(* PLC project CodesysTest.project, PN2IC PLCopen CODESYS V3.5 SP17 Patch 3 *)
(* stored: creationDateTime 2023-02-26T17:02:07, modificationDateTime 2023-02-26T17:02:07 *)

PROGRAM flow_1

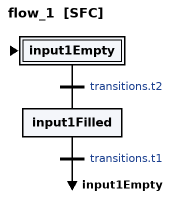
INITIAL_STEP input1Empty:
END_STEP
TRANSITION FROM input1Empty TO input1Filled
  := transitions.t2;
END_TRANSITION
STEP input1Filled:
END_STEP
TRANSITION FROM input1Filled TO input1Empty
  := transitions.t1;
END_TRANSITION
END_PROGRAM

PROGRAM flow_11

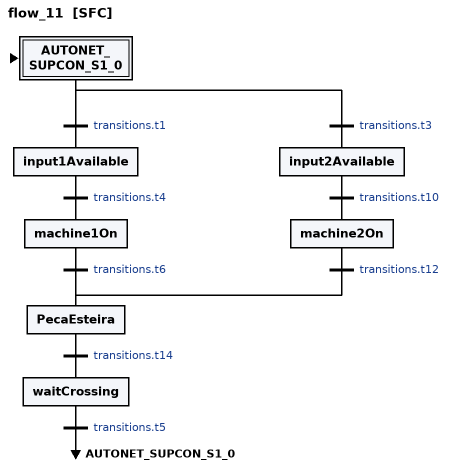
INITIAL_STEP AUTONET_SUPCON_S1_0:
END_STEP
TRANSITION FROM AUTONET_SUPCON_S1_0 TO input1Available
  := transitions.t1;
END_TRANSITION
TRANSITION FROM AUTONET_SUPCON_S1_0 TO input2Available
  := transitions.t3;
END_TRANSITION
STEP input1Available:
END_STEP
TRANSITION FROM input1Available TO machine1On
  := transitions.t4;
END_TRANSITION
STEP machine1On:
END_STEP
TRANSITION FROM machine1On TO PecaEsteira
  := transitions.t6;
END_TRANSITION
STEP input2Available:
END_STEP
TRANSITION FROM input2Available TO machine2On
  := transitions.t10;
END_TRANSITION
STEP machine2On:
END_STEP
TRANSITION FROM machine2On TO PecaEsteira
  := transitions.t12;
END_TRANSITION
STEP PecaEsteira:
END_STEP
TRANSITION FROM PecaEsteira TO waitCrossing
  := transitions.t14;
END_TRANSITION
STEP waitCrossing:
END_STEP
TRANSITION FROM waitCrossing TO AUTONET_SUPCON_S1_0
  := transitions.t5;
END_TRANSITION
END_PROGRAM

PROGRAM flow_12

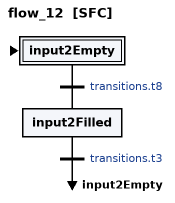
INITIAL_STEP input2Empty:
END_STEP
TRANSITION FROM input2Empty TO input2Filled
  := transitions.t8;
END_TRANSITION
STEP input2Filled:
END_STEP
TRANSITION FROM input2Filled TO input2Empty
  := transitions.t3;
END_TRANSITION
END_PROGRAM

PROGRAM flow_9

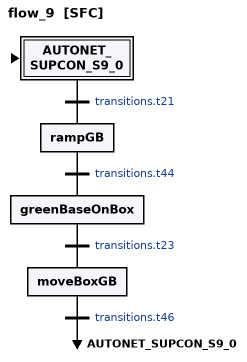
INITIAL_STEP AUTONET_SUPCON_S9_0:
END_STEP
TRANSITION FROM AUTONET_SUPCON_S9_0 TO rampGB
  := transitions.t21;
END_TRANSITION
STEP rampGB:
END_STEP
TRANSITION FROM rampGB TO greenBaseOnBox
  := transitions.t44;
END_TRANSITION
STEP greenBaseOnBox:
END_STEP
TRANSITION FROM greenBaseOnBox TO moveBoxGB
  := transitions.t23;
END_TRANSITION
STEP moveBoxGB:
END_STEP
TRANSITION FROM moveBoxGB TO AUTONET_SUPCON_S9_0
  := transitions.t46;
END_TRANSITION
END_PROGRAM

PROGRAM flow_3

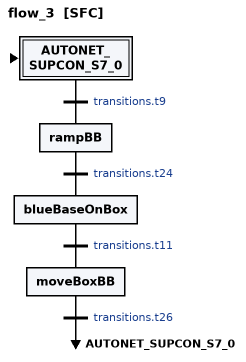
INITIAL_STEP AUTONET_SUPCON_S7_0:
END_STEP
TRANSITION FROM AUTONET_SUPCON_S7_0 TO rampBB
  := transitions.t9;
END_TRANSITION
STEP rampBB:
END_STEP
TRANSITION FROM rampBB TO blueBaseOnBox
  := transitions.t24;
END_TRANSITION
STEP blueBaseOnBox:
END_STEP
TRANSITION FROM blueBaseOnBox TO moveBoxBB
  := transitions.t11;
END_TRANSITION
STEP moveBoxBB:
END_STEP
TRANSITION FROM moveBoxBB TO AUTONET_SUPCON_S7_0
  := transitions.t26;
END_TRANSITION
END_PROGRAM

PROGRAM flow_15

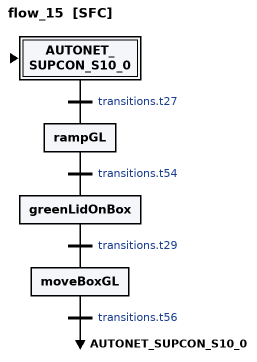
INITIAL_STEP AUTONET_SUPCON_S10_0:
END_STEP
TRANSITION FROM AUTONET_SUPCON_S10_0 TO rampGL
  := transitions.t27;
END_TRANSITION
STEP rampGL:
END_STEP
TRANSITION FROM rampGL TO greenLidOnBox
  := transitions.t54;
END_TRANSITION
STEP greenLidOnBox:
END_STEP
TRANSITION FROM greenLidOnBox TO moveBoxGL
  := transitions.t29;
END_TRANSITION
STEP moveBoxGL:
END_STEP
TRANSITION FROM moveBoxGL TO AUTONET_SUPCON_S10_0
  := transitions.t56;
END_TRANSITION
END_PROGRAM

PROGRAM flow_4

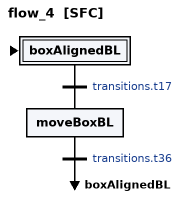
INITIAL_STEP boxAlignedBL:
END_STEP
TRANSITION FROM boxAlignedBL TO moveBoxBL
  := transitions.t17;
END_TRANSITION
STEP moveBoxBL:
END_STEP
TRANSITION FROM moveBoxBL TO boxAlignedBL
  := transitions.t36;
END_TRANSITION
END_PROGRAM

PROGRAM flow_5

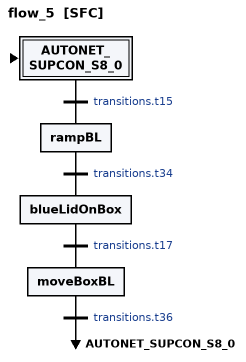
INITIAL_STEP AUTONET_SUPCON_S8_0:
END_STEP
TRANSITION FROM AUTONET_SUPCON_S8_0 TO rampBL
  := transitions.t15;
END_TRANSITION
STEP rampBL:
END_STEP
TRANSITION FROM rampBL TO blueLidOnBox
  := transitions.t34;
END_TRANSITION
STEP blueLidOnBox:
END_STEP
TRANSITION FROM blueLidOnBox TO moveBoxBL
  := transitions.t17;
END_TRANSITION
STEP moveBoxBL:
END_STEP
TRANSITION FROM moveBoxBL TO AUTONET_SUPCON_S8_0
  := transitions.t36;
END_TRANSITION
END_PROGRAM

PROGRAM flow_8

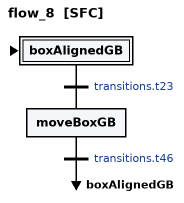
INITIAL_STEP boxAlignedGB:
END_STEP
TRANSITION FROM boxAlignedGB TO moveBoxGB
  := transitions.t23;
END_TRANSITION
STEP moveBoxGB:
END_STEP
TRANSITION FROM moveBoxGB TO boxAlignedGB
  := transitions.t46;
END_TRANSITION
END_PROGRAM

PROGRAM flow_6

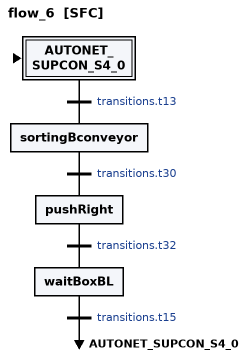
INITIAL_STEP AUTONET_SUPCON_S4_0:
END_STEP
TRANSITION FROM AUTONET_SUPCON_S4_0 TO sortingBconveyor
  := transitions.t13;
END_TRANSITION
STEP sortingBconveyor:
END_STEP
TRANSITION FROM sortingBconveyor TO pushRight
  := transitions.t30;
END_TRANSITION
STEP pushRight:
END_STEP
TRANSITION FROM pushRight TO waitBoxBL
  := transitions.t32;
END_TRANSITION
STEP waitBoxBL:
END_STEP
TRANSITION FROM waitBoxBL TO AUTONET_SUPCON_S4_0
  := transitions.t15;
END_TRANSITION
END_PROGRAM

PROGRAM flow_10

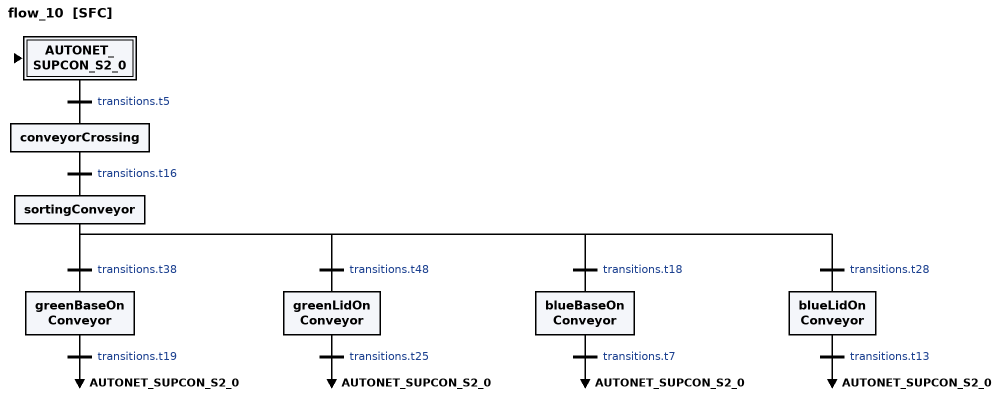
INITIAL_STEP AUTONET_SUPCON_S2_0:
END_STEP
TRANSITION FROM AUTONET_SUPCON_S2_0 TO conveyorCrossing
  := transitions.t5;
END_TRANSITION
STEP conveyorCrossing:
END_STEP
TRANSITION FROM conveyorCrossing TO sortingConveyor
  := transitions.t16;
END_TRANSITION
STEP sortingConveyor:
END_STEP
TRANSITION FROM sortingConveyor TO greenBaseOnConveyor
  := transitions.t38;
END_TRANSITION
TRANSITION FROM sortingConveyor TO greenLidOnConveyor
  := transitions.t48;
END_TRANSITION
TRANSITION FROM sortingConveyor TO blueBaseOnConveyor
  := transitions.t18;
END_TRANSITION
TRANSITION FROM sortingConveyor TO blueLidOnConveyor
  := transitions.t28;
END_TRANSITION
STEP greenBaseOnConveyor:
END_STEP
TRANSITION FROM greenBaseOnConveyor TO AUTONET_SUPCON_S2_0
  := transitions.t19;
END_TRANSITION
STEP greenLidOnConveyor:
END_STEP
TRANSITION FROM greenLidOnConveyor TO AUTONET_SUPCON_S2_0
  := transitions.t25;
END_TRANSITION
STEP blueBaseOnConveyor:
END_STEP
TRANSITION FROM blueBaseOnConveyor TO AUTONET_SUPCON_S2_0
  := transitions.t7;
END_TRANSITION
STEP blueLidOnConveyor:
END_STEP
TRANSITION FROM blueLidOnConveyor TO AUTONET_SUPCON_S2_0
  := transitions.t13;
END_TRANSITION
END_PROGRAM

PROGRAM flow_2

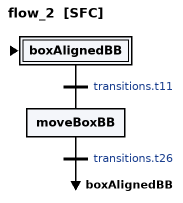
INITIAL_STEP boxAlignedBB:
END_STEP
TRANSITION FROM boxAlignedBB TO moveBoxBB
  := transitions.t11;
END_TRANSITION
STEP moveBoxBB:
END_STEP
TRANSITION FROM moveBoxBB TO boxAlignedBB
  := transitions.t26;
END_TRANSITION
END_PROGRAM

PROGRAM flow_13

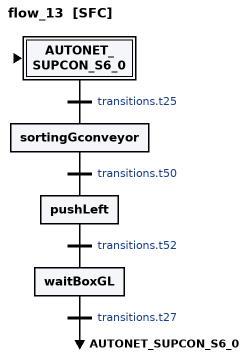
INITIAL_STEP AUTONET_SUPCON_S6_0:
END_STEP
TRANSITION FROM AUTONET_SUPCON_S6_0 TO sortingGconveyor
  := transitions.t25;
END_TRANSITION
STEP sortingGconveyor:
END_STEP
TRANSITION FROM sortingGconveyor TO pushLeft
  := transitions.t50;
END_TRANSITION
STEP pushLeft:
END_STEP
TRANSITION FROM pushLeft TO waitBoxGL
  := transitions.t52;
END_TRANSITION
STEP waitBoxGL:
END_STEP
TRANSITION FROM waitBoxGL TO AUTONET_SUPCON_S6_0
  := transitions.t27;
END_TRANSITION
END_PROGRAM

PROGRAM flow_14

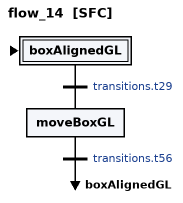
INITIAL_STEP boxAlignedGL:
END_STEP
TRANSITION FROM boxAlignedGL TO moveBoxGL
  := transitions.t29;
END_TRANSITION
STEP moveBoxGL:
END_STEP
TRANSITION FROM moveBoxGL TO boxAlignedGL
  := transitions.t56;
END_TRANSITION
END_PROGRAM

PROGRAM flow_16

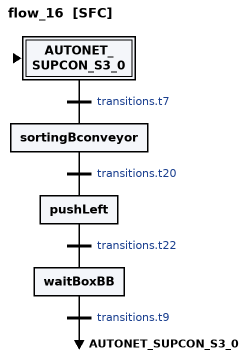
INITIAL_STEP AUTONET_SUPCON_S3_0:
END_STEP
TRANSITION FROM AUTONET_SUPCON_S3_0 TO sortingBconveyor
  := transitions.t7;
END_TRANSITION
STEP sortingBconveyor:
END_STEP
TRANSITION FROM sortingBconveyor TO pushLeft
  := transitions.t20;
END_TRANSITION
STEP pushLeft:
END_STEP
TRANSITION FROM pushLeft TO waitBoxBB
  := transitions.t22;
END_TRANSITION
STEP waitBoxBB:
END_STEP
TRANSITION FROM waitBoxBB TO AUTONET_SUPCON_S3_0
  := transitions.t9;
END_TRANSITION
END_PROGRAM

PROGRAM flow_7

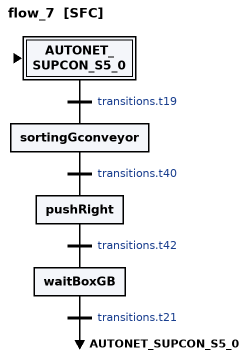
INITIAL_STEP AUTONET_SUPCON_S5_0:
END_STEP
TRANSITION FROM AUTONET_SUPCON_S5_0 TO sortingGconveyor
  := transitions.t19;
END_TRANSITION
STEP sortingGconveyor:
END_STEP
TRANSITION FROM sortingGconveyor TO pushRight
  := transitions.t40;
END_TRANSITION
STEP pushRight:
END_STEP
TRANSITION FROM pushRight TO waitBoxGB
  := transitions.t42;
END_TRANSITION
STEP waitBoxGB:
END_STEP
TRANSITION FROM waitBoxGB TO AUTONET_SUPCON_S5_0
  := transitions.t21;
END_TRANSITION
END_PROGRAM

PROGRAM transitions

         
        
END_PROGRAM

CONFIGURATION Application
  RESOURCE Application ON PLC
    VAR_GLOBAL  (* GVL *)
      t44 : BOOL;
      t46 : BOOL;
      t48 : BOOL;
      t5 : BOOL;
      t50 : BOOL;
      t52 : BOOL;
      t54 : BOOL;
      t56 : BOOL;
      t6 : BOOL;
      t7 : BOOL;
      t8 : BOOL;
      t9 : BOOL;
      t1 : BOOL;
      t10 : BOOL;
      t11 : BOOL;
      t12 : BOOL;
      t13 : BOOL;
      t14 : BOOL;
      t15 : BOOL;
      t16 : BOOL;
      t17 : BOOL;
      t18 : BOOL;
      t19 : BOOL;
      t2 : BOOL;
      t20 : BOOL;
      t21 : BOOL;
      t22 : BOOL;
      t23 : BOOL;
      t24 : BOOL;
      t25 : BOOL;
      t26 : BOOL;
      t27 : BOOL;
      t28 : BOOL;
      t29 : BOOL;
      t3 : BOOL;
      t30 : BOOL;
      t32 : BOOL;
      t34 : BOOL;
      t36 : BOOL;
      t38 : BOOL;
      t4 : BOOL;
      t40 : BOOL;
      t42 : BOOL;
    END_VAR
    TASK MainTask(INTERVAL := T#20ms, PRIORITY := 1);
    PROGRAM flow_1 WITH MainTask : flow_1;
    PROGRAM flow_11 WITH MainTask : flow_11;
    PROGRAM flow_12 WITH MainTask : flow_12;
    PROGRAM flow_9 WITH MainTask : flow_9;
    PROGRAM flow_3 WITH MainTask : flow_3;
    PROGRAM flow_15 WITH MainTask : flow_15;
    PROGRAM flow_4 WITH MainTask : flow_4;
    PROGRAM flow_5 WITH MainTask : flow_5;
    PROGRAM flow_8 WITH MainTask : flow_8;
    PROGRAM flow_6 WITH MainTask : flow_6;
    PROGRAM flow_10 WITH MainTask : flow_10;
    PROGRAM flow_2 WITH MainTask : flow_2;
    PROGRAM flow_13 WITH MainTask : flow_13;
    PROGRAM flow_14 WITH MainTask : flow_14;
    PROGRAM flow_16 WITH MainTask : flow_16;
    PROGRAM flow_7 WITH MainTask : flow_7;
  END_RESOURCE
END_CONFIGURATION
